FUNCTION_BLOCK POU
VAR_INPUT
	bExecute		: BOOL;
END_VAR
VAR_OUTPUT
	bDone			: BOOL;
	bError			: BOOL;
	wErrorID		: BOOL;
END_VAR
VAR
	
END_VAR

END_FUNCTION_BLOCK

(* stored: Version 1.1.0.1, ProductVersion 3.1.4024.11
   POU POU: Id {d068a546-df5c-4264-9970-4623701827c7}, SpecialFunc None *)
